{attribute 'qualified_only'}
VAR_GLOBAL CONSTANT
	COMP_CAP		: UDINT;
END_VAR

(* stored: Version 1.1.0.1
   GVL Param: Id {9432ed60-25e9-4a8c-976b-8360a4b35775}, ParameterList True *)
